FUNCTION_BLOCK PRODUCTION_SCHEDULER (* Composite Function Block Type *)
  (* Standard: 61499-2 *)
  (* Version 0.0, 12/17/2022, Dmitrii, Flexbridge AB, template *)
  PACKAGE Main;
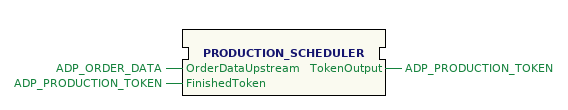
  SOCKETS
    OrderDataUpstream : ADP_ORDER_DATA;
    FinishedToken : ADP_PRODUCTION_TOKEN;
  END_SOCKETS
  PLUGS
    TokenOutput : ADP_PRODUCTION_TOKEN;
  END_PLUGS
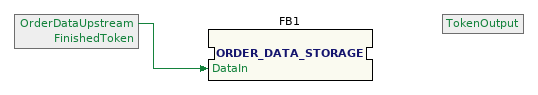
  FBS
    FB1 : ORDER_DATA_STORAGE;
  END_FBS
  ADAPTER_CONNECTIONS
    OrderDataUpstream TO FB1.DataIn;
  END_CONNECTIONS
END_FUNCTION_BLOCK
